// TIA Portal V19 export
FUNCTION_BLOCK "TYPIC_C104_IF_KLP"   // FB94, FBD
TITLE = TYPIC_C104_IF_KLP: Brandstofklep
{ S7_Optimized_Access := 'TRUE' }
AUTHOR : OCOTECH
FAMILY : Typical
NAME : C104.705
// Logisch Object Besturing: C104.705
// 
// De interne functie Brandstofklep verzorgt de bewaking van een brandstofklep van een noodstroomaggregaat.
// stored: MemoryReserve 10, SetENOAutomatically false
   VAR_INPUT
      EXT_AUT { ExternalAccessible := 'False'; ExternalVisible := 'False'; ExternalWritable := 'False'} : Bool;   // Externe (hoofd) beveiliging (1 = OK)
      EXT_HW { ExternalAccessible := 'False'; ExternalVisible := 'False'; ExternalWritable := 'False'} : Bool;   // Sturings hardware (PLC) bewaking (1 = OK)
      IN_STO_NOK { ExternalAccessible := 'False'; ExternalVisible := 'False'; ExternalWritable := 'False'} : Bool;   // Storing aanwezig die niet observeerbaar tot gevolg heeft
      IN_STO_OK { ExternalAccessible := 'False'; ExternalVisible := 'False'; ExternalWritable := 'False'} : Bool;   // Storing aanwezig die observeerbaarheid niet beinvloed
      IN_OPEN { ExternalAccessible := 'False'; ExternalVisible := 'False'; ExternalWritable := 'False'} : Bool;   // Brandstofklep open
      IN_TOE { ExternalAccessible := 'False'; ExternalVisible := 'False'; ExternalWritable := 'False'} : Bool;   // Brandstofklep dicht
      IN_AUT_C104 { ExternalAccessible := 'False'; ExternalVisible := 'False'; ExternalWritable := 'False'} : Bool;   // Beveiligingen: serie geschakelde terugmelding (1 = OK)
   END_VAR
   VAR_OUTPUT
      VAR_IF_KLP { ExternalAccessible := 'False'; ExternalVisible := 'False'; ExternalWritable := 'False'} : "C104_VAR_IF_KLP_TYPIC";   // Struct met alle variabelen naar bovenliggende functies
   END_VAR
   VAR
      STO { ExternalWritable := 'False'} : Struct   // Storingen
         A001 : Bool;   // Beveiliging aangesproken
         A002 : Bool;   // Brandstofklep in storing
         A003 : Bool;   // Algemene storing brandstofklep
      END_STRUCT;
      VAR { ExternalWritable := 'False'} : Struct   // Variabelen
         OPEN { ExternalAccessible := 'False'; ExternalVisible := 'False'} : Bool;   // Brandstofklep open
         TOE { ExternalAccessible := 'False'; ExternalVisible := 'False'} : Bool;   // Brandstofklep dicht
         EXT_AUT { ExternalAccessible := 'False'; ExternalVisible := 'False'} : Bool;   // Externe (hoofd) beveiliging aangesproken
         EXT_HW { ExternalAccessible := 'False'; ExternalVisible := 'False'} : Bool;   // Sturings hardware (PLC) in storing
      END_STRUCT;
   END_VAR
BEGIN

REGION Network 1: START
END_REGION

REGION Network 2: +++ Verwerking statussen +++
   // Bepalen van de statussen van de brandstofklep.
END_REGION

REGION Network 3: +++ Storingen +++
   // Verwerken van de storingsmeldingen (inputs).
END_REGION

REGION Network 4: Storing A001: Beveiliging aangesproken
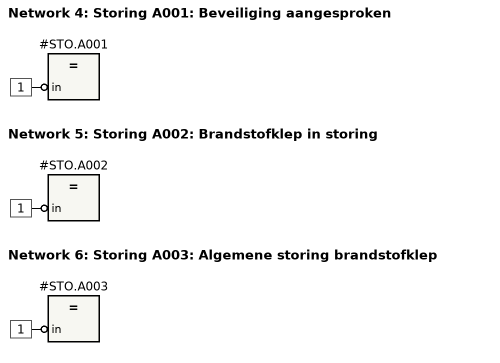
   #STO.A001 := NOT 1;
END_REGION

REGION Network 5: Storing A002: Brandstofklep in storing
   #STO.A002 := NOT 1;
END_REGION

REGION Network 6: Storing A003: Algemene storing brandstofklep
   #STO.A003 := NOT 1;
END_REGION

REGION Network 7 (SCL): EINDE
   // Variabelen van intern scada rakvlak naar outputs copieren
   #VAR_IF_KLP.OPEN := #VAR.OPEN;
   #VAR_IF_KLP.TOE := #VAR.TOE;
   #VAR_IF_KLP.EXT_AUT := #VAR.EXT_AUT;
   #VAR_IF_KLP.EXT_HW := #VAR.EXT_HW;
   #VAR_IF_KLP.STO := #STO;
END_REGION
END_FUNCTION_BLOCK
